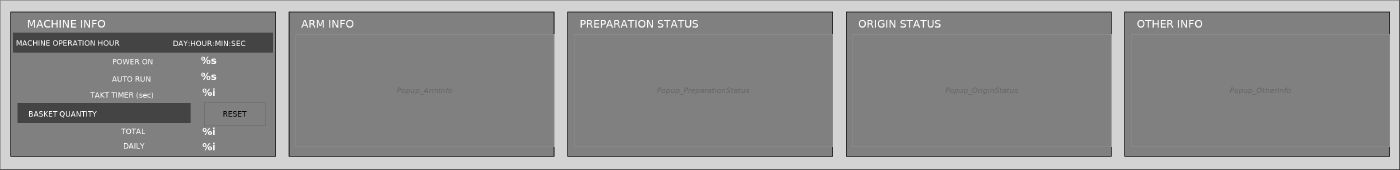
VISUALIZATION Popup_AllInfo  // 1920x234
    Rectangle (0,0 1920x234)
    RoundedRectangle (14,16 364x199)
    Rectangle (18,45 356x27)
    Label (19,44 183x31), "MACHINE OPERATION HOUR"
    Label (45,73 168x24), "POWER ON"
    Label (44,97 166x24), "AUTO RUN"
    Label (48,119 166x24), "TAKT TIMER (sec)"
    Label (42,169 160x24), "TOTAL"
    Label (50,189 151x24), "DAILY"
    Button (280,141 84x32), "RESET", colour toggle: bBasketTotalizerResetPB_Daily
        tap bBasketTotalizerResetPB_Daily
        OnMouseClick: change screen: AutoMain_Page
    Rectangle (24,142 237x27)
    Label (36,145 134x24), "BASKET QUANTITY"
    Label (34,21 319x24), "MACHINE INFO"
    RoundedRectangle (396,16 364x199)
    Frame (405,47 355x155)
        shows Popup_ArmInfo()
    Label (410,21 330x24), "ARM INFO"
    RoundedRectangle (778,16 364x199)
    Frame (787,47 355x155)
        shows Popup_PreparationStatus()
    Label (792,21 202x24), "PREPARATION STATUS"
    Group (1160,16 364x199)
        RoundedRectangle (0,0 364x199)
        Frame (9,31 355x155)
            shows Popup_OriginStatus()
        Label (14,5 173x24), "ORIGIN STATUS"
    RoundedRectangle (1542,16 364x199)
    Frame (1551,47 355x155)
        shows Popup_OtherInfo()
    Label (1556,21 306x24), "OTHER INFO"
    Label (213,76 38x22)
    Rectangle (202,75 169x17), "%s", text variable: sMachineOnTime_Customer
    Label (203,48 168x24), "DAY:HOUR:MIN:SEC"
    Rectangle (202,97 169x17), "%s", text variable: sMachineRunningTime_Customer
    Rectangle (202,119 169x17), "%i", text variable: iActTactTime
    Rectangle (202,173 169x17), "%i", text variable: diTotalBasketQty_Customer
    Rectangle (202,194 169x17), "%i", text variable: diTotalBasketQty_Daily
END_VISUALIZATION

(* stored: Version 1.1.0.1, ProductVersion 3.1.4024.12
   Visu Popup_AllInfo: Id {88e7be81-0201-41f2-8be6-259ce6bea796} *)
